FUNCTION_BLOCK AutoModeSteam (* Composite Function Block Type *)
  (* Standard: 61499-2 *)
  (* Version 0.0, 2011-12-29, 4DIAC-IDE, 4DIAC-Consortium *)
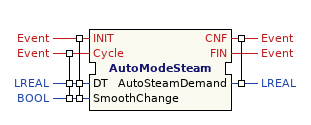
  EVENT_INPUT
    INIT WITH DT, SmoothChange; (* Initialization Request *)
    Cycle WITH DT, SmoothChange; (* Normal Execution Request *)
  END_EVENT
  EVENT_OUTPUT
    CNF WITH AutoSteamDemand; (* Execution Confirmation *)
    FIN;
  END_EVENT
  VAR_INPUT
    DT : LREAL; (* Input event qualifier *)
    SmoothChange : BOOL := 1;
  END_VAR
  VAR_OUTPUT
    AutoSteamDemand : LREAL; (* Output event qualifier *)
  END_VAR
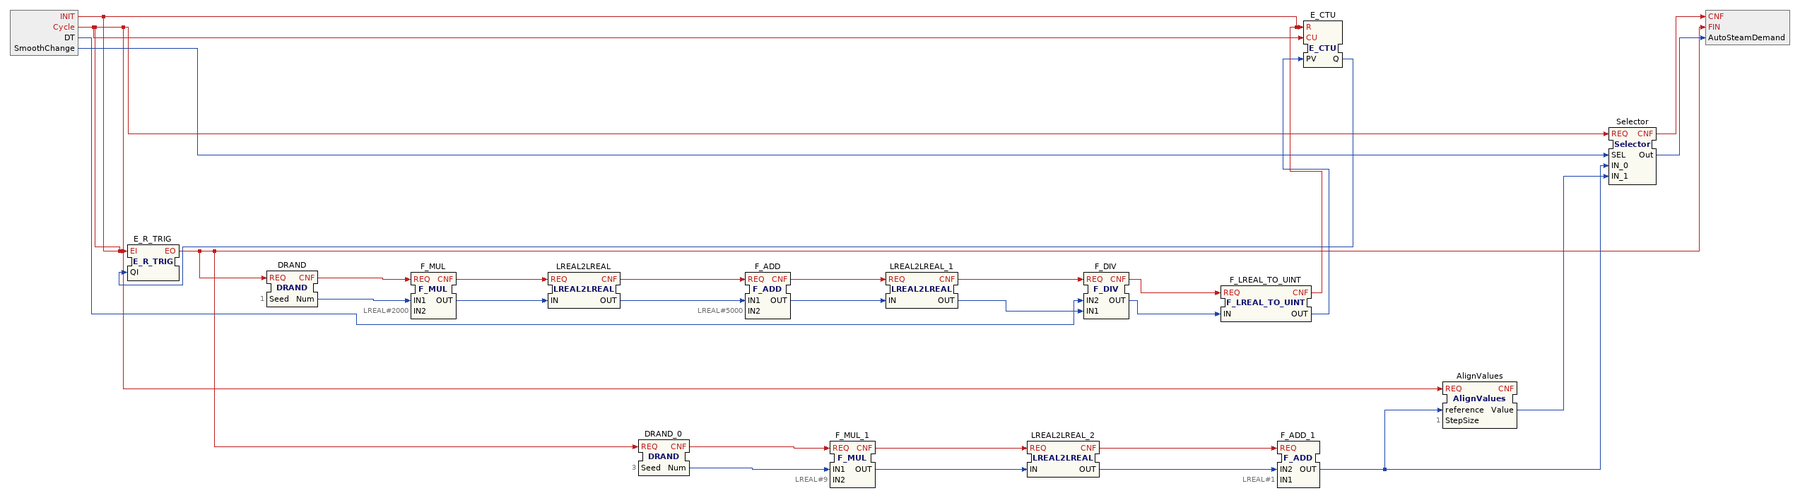
  FBS
    E_CTU : E_CTU;
    E_R_TRIG : E_R_TRIG;
    DRAND : DRAND(Seed := 1);
    F_LREAL_TO_UINT : F_LREAL_TO_UINT;
    DRAND_0 : DRAND(Seed := 3);
    AlignValues : AlignValues(StepSize := 1);
    Selector : Selector;
    F_MUL : F_MUL(IN2 := LREAL#2000);
    F_ADD : F_ADD(IN2 := LREAL#5000);
    F_DIV : F_DIV;
    LREAL2LREAL : LREAL2LREAL;
    LREAL2LREAL_1 : LREAL2LREAL;
    F_MUL_1 : F_MUL(IN2 := LREAL#9);
    F_ADD_1 : F_ADD(IN1 := LREAL#1);
    LREAL2LREAL_2 : LREAL2LREAL;
  END_FBS
  EVENT_CONNECTIONS
    F_LREAL_TO_UINT.CNF TO E_CTU.R;
    Cycle TO E_CTU.CU;
    E_R_TRIG.EO TO DRAND.REQ;
    INIT TO E_R_TRIG.EI;
    INIT TO E_CTU.R;
    E_R_TRIG.EO TO DRAND_0.REQ;
    Cycle TO E_R_TRIG.EI;
    Cycle TO AlignValues.REQ;
    Cycle TO Selector.REQ;
    Selector.CNF TO CNF;
    E_R_TRIG.EO TO FIN;
    DRAND.CNF TO F_MUL.REQ;
    F_MUL.CNF TO LREAL2LREAL.REQ;
    LREAL2LREAL.CNF TO F_ADD.REQ;
    F_ADD.CNF TO LREAL2LREAL_1.REQ;
    LREAL2LREAL_1.CNF TO F_DIV.REQ;
    F_DIV.CNF TO F_LREAL_TO_UINT.REQ;
    LREAL2LREAL_2.CNF TO F_ADD_1.REQ;
    F_MUL_1.CNF TO LREAL2LREAL_2.REQ;
    DRAND_0.CNF TO F_MUL_1.REQ;
  END_CONNECTIONS
  DATA_CONNECTIONS
    F_LREAL_TO_UINT.OUT TO E_CTU.PV;
    E_CTU.Q TO E_R_TRIG.QI;
    SmoothChange TO Selector.SEL;
    AlignValues.Value TO Selector.IN_1;
    Selector.Out TO AutoSteamDemand;
    DRAND.Num TO F_MUL.IN1;
    DT TO F_DIV.IN2;
    F_MUL.OUT TO LREAL2LREAL.IN;
    LREAL2LREAL.OUT TO F_ADD.IN1;
    F_ADD.OUT TO LREAL2LREAL_1.IN;
    LREAL2LREAL_1.OUT TO F_DIV.IN1;
    F_DIV.OUT TO F_LREAL_TO_UINT.IN;
    F_ADD_1.OUT TO Selector.IN_0;
    F_ADD_1.OUT TO AlignValues.reference;
    LREAL2LREAL_2.OUT TO F_ADD_1.IN2;
    F_MUL_1.OUT TO LREAL2LREAL_2.IN;
    DRAND_0.Num TO F_MUL_1.IN1;
  END_CONNECTIONS
END_FUNCTION_BLOCK
